KUKA KRL program: GETPOINT.src

&ACCESS RVP1
&REL 33
&PARAM TEMPLATE = C:\KRC\Roboter\Template\FunctionVorgabe
&PARAM EDITMASK = *
DEFFCT FRAME GETPOINT(DIRECTION:IN, SIGN:IN)
DECL FRAME POINT
CHAR DIRECTION
INT SIGN
$TOOL=TOOL_DATA[5]
$ORI_TYPE=#CONSTANT
$TOOL=TOOL_DATA[5]
$VEL.CP=1.0
$VEL.ORI1=100
$VEL.ORI2=100
$ACC.CP=1.0
$ACC.ORI1=100
$ACC.ORI2=100

POINT.A=0.0
POINT.B=0.0
POINT.C=-180
POINT.Z=50
IF DIRECTION=="Z" THEN
  POINT.X=12.24
  POINT.Y=-591.6
  POINT.Z=65.39
ENDIF
IF DIRECTION=="X" THEN
  POINT.Y=-592.02
  IF SIGN==1 THEN
    POINT.X=-25.7
  ENDIF
  IF SIGN==-1 THEN
    POINT.X=49.8
  ENDIF
ENDIF
IF DIRECTION=="Y" THEN
  POINT.X=15
  IF SIGN==1 THEN
    POINT.Y=-629.3
  ENDIF
  IF SIGN==-1 THEN
    POINT.Y=-555
  ENDIF
ENDIF
RETURN POINT
ENDFCT
